// TIA Portal V16 export
// export: Created 2022-02-11T14:39:19.0580215Z, ExportSetting WithDefaults, DisplayName Totally Integrated Automation Portal, DisplayVersion V16 Update 1, DisplayName TIA Portal Version Control Interface, DisplayVersion V16, DisplayName TIA Portal Openness, DisplayVersion V16, DisplayName SINAMICS Startdrive Advanced, DisplayVersion V16 Update 5, DisplayName SINAMICS Startdrive G130, G150, S120, S150, SINAMICS MV, S210, DisplayVersion V16 Update 5, DisplayName SINAMICS Startdrive G110M, G120, G120C, G120D, G120P, G115D, DisplayVersion V16 Update 5, DisplayName STEP 7 Professional, DisplayVersion V16, DisplayName STEP 7 Safety, DisplayVersion V16, DisplayName WinCC Advanced, DisplayVersion V16, DisplayName SIMATIC Visualization Architect, DisplayVersion V16
ORGANIZATION_BLOCK "Main"   // OB1, LAD, ProgramCycle
TITLE = "Main Program Sweep (Cycle)"
VERSION : 0.1
// stored: IsIECCheckEnabled false
   VAR_TEMP
      OB1_EV_CLASS : Byte;   // Bits 0-3 = 1 (Coming event), Bits 4-7 = 1 (Event class 1)
      OB1_SCAN_1 : Byte;   // 1 (Cold restart scan 1 of OB 1), 3 (Scan 2-n of OB 1)
      OB1_PRIORITY : Byte;   // Priority of OB Execution
      OB1_OB_NUMBR : Byte;   // 1 (Organization block 1, OB1)
      OB1_RESERVED_1 : Byte;   // Reserved for system
      OB1_RESERVED_2 : Byte;   // Reserved for system
      BoardPosition : Int;   // Позиция подвижного борта
      OB1_PREV_CYCLE : Int;   // Cycle time of previous OB1 scan (milliseconds)
      OB1_MIN_CYCLE : Int;   // Minimum cycle time of OB1 (milliseconds)
      OB1_MAX_CYCLE : Int;   // Maximum cycle time of OB1 (milliseconds)
      OB1_DATE_TIME : Date_And_Time;   // Date and time OB1 started
   END_VAR
   VAR_TEMP   // added for the SCL form of the ladder/FBD networks
      _w1 : Bool;
      _w2 : Bool;
      _w3 : Bool;
      _s5time1 : S5Time;
   END_VAR
BEGIN

REGION Network 1: ProcessInput
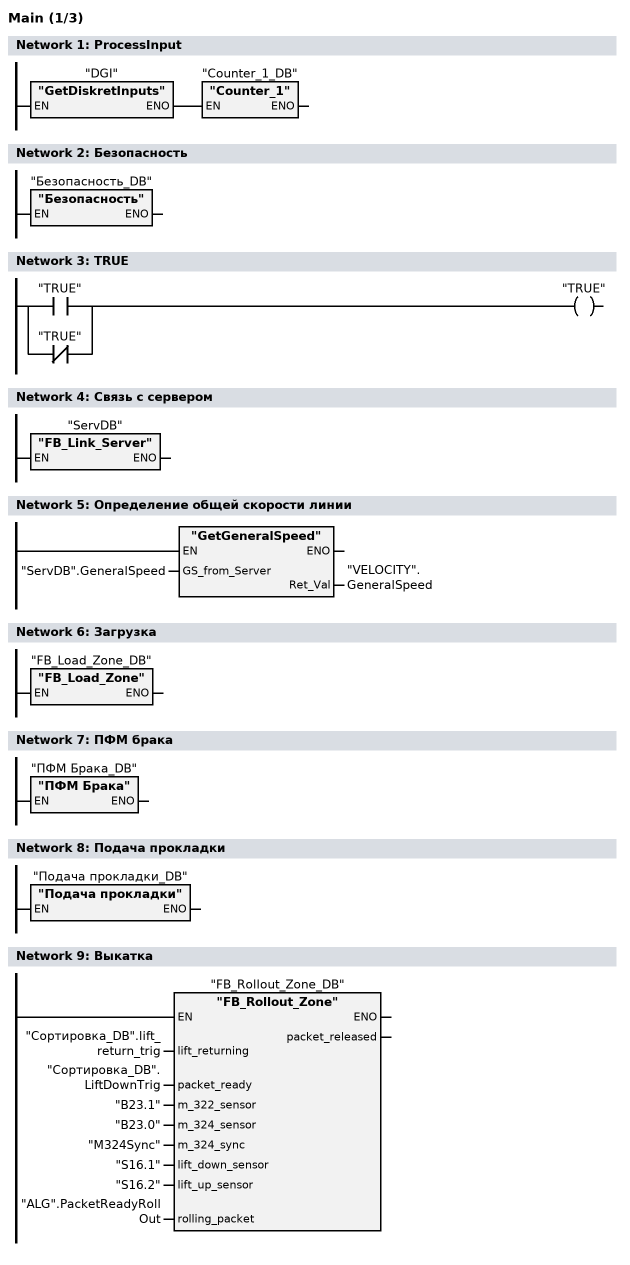
   RUNG wire#powerrail
      "DGI"()
      "Counter_1_DB"()
   END_RUNG
   // the same network as SCL:
   "DGI"(ENO => #_w1);   // "GetDiskretInputs"
   IF #_w1 THEN
       "Counter_1_DB"();   // "Counter_1"
   END_IF;
END_REGION

REGION Network 2: Безопасность
   RUNG wire#powerrail
      "Безопасность_DB"()
   END_RUNG
   // the same network as SCL:
   "Безопасность_DB"();   // "Безопасность"
END_REGION

REGION Network 3: TRUE
   RUNG wire#powerrail
      Contact( "TRUE" )
      wire#w1
      Coil( "TRUE" )
   END_RUNG
   RUNG wire#powerrail
      I_Contact( "TRUE" )
   END_RUNG wire#w1
   // the same network as SCL:
   "TRUE" := "TRUE" OR NOT "TRUE";
END_REGION

REGION Network 4: Связь с сервером
   RUNG wire#powerrail
      "ServDB"()
   END_RUNG
   // the same network as SCL:
   "ServDB"();   // "FB_Link_Server"
END_REGION

REGION Network 5: Определение общей скорости линии
   RUNG wire#powerrail
      "GetGeneralSpeed"(GS_from_Server := "ServDB".GeneralSpeed, Ret_Val => "VELOCITY".GeneralSpeed)
   END_RUNG
   // the same network as SCL:
   "VELOCITY".GeneralSpeed := "GetGeneralSpeed"(GS_from_Server := "ServDB".GeneralSpeed);
END_REGION

REGION Network 6: Загрузка
   RUNG wire#powerrail
      "FB_Load_Zone_DB"()
   END_RUNG
   // the same network as SCL:
   "FB_Load_Zone_DB"();   // "FB_Load_Zone"
END_REGION

REGION Network 7: ПФМ брака
   RUNG wire#powerrail
      "ПФМ Брака_DB"()
   END_RUNG
   // the same network as SCL:
   "ПФМ Брака_DB"();   // "ПФМ Брака"
END_REGION

REGION Network 8: Подача прокладки
   RUNG wire#powerrail
      "Подача прокладки_DB"()
   END_RUNG
   // the same network as SCL:
   "Подача прокладки_DB"();   // "Подача прокладки"
END_REGION

REGION Network 9: Выкатка
   RUNG wire#powerrail
      "FB_Rollout_Zone_DB"(lift_returning := "Сортировка_DB".lift_return_trig, packet_ready := "Сортировка_DB".LiftDownTrig, m_322_sensor := "B23.1", m_324_sensor := "B23.0", m_324_sync := "M324Sync", lift_down_sensor := "S16.1", lift_up_sensor := "S16.2", rolling_packet := "ALG".PacketReadyRollOut, packet_released =>)
   END_RUNG
   // the same network as SCL:
   "FB_Rollout_Zone_DB"(lift_returning := "Сортировка_DB".lift_return_trig,   // "FB_Rollout_Zone"
                        packet_ready := "Сортировка_DB".LiftDownTrig,
                        m_322_sensor := "B23.1",
                        m_324_sensor := "B23.0",
                        m_324_sync := "M324Sync",
                        lift_down_sensor := "S16.1",
                        lift_up_sensor := "S16.2",
                        rolling_packet := "ALG".PacketReadyRollOut);
END_REGION

REGION Network 10: Карусель прокладок
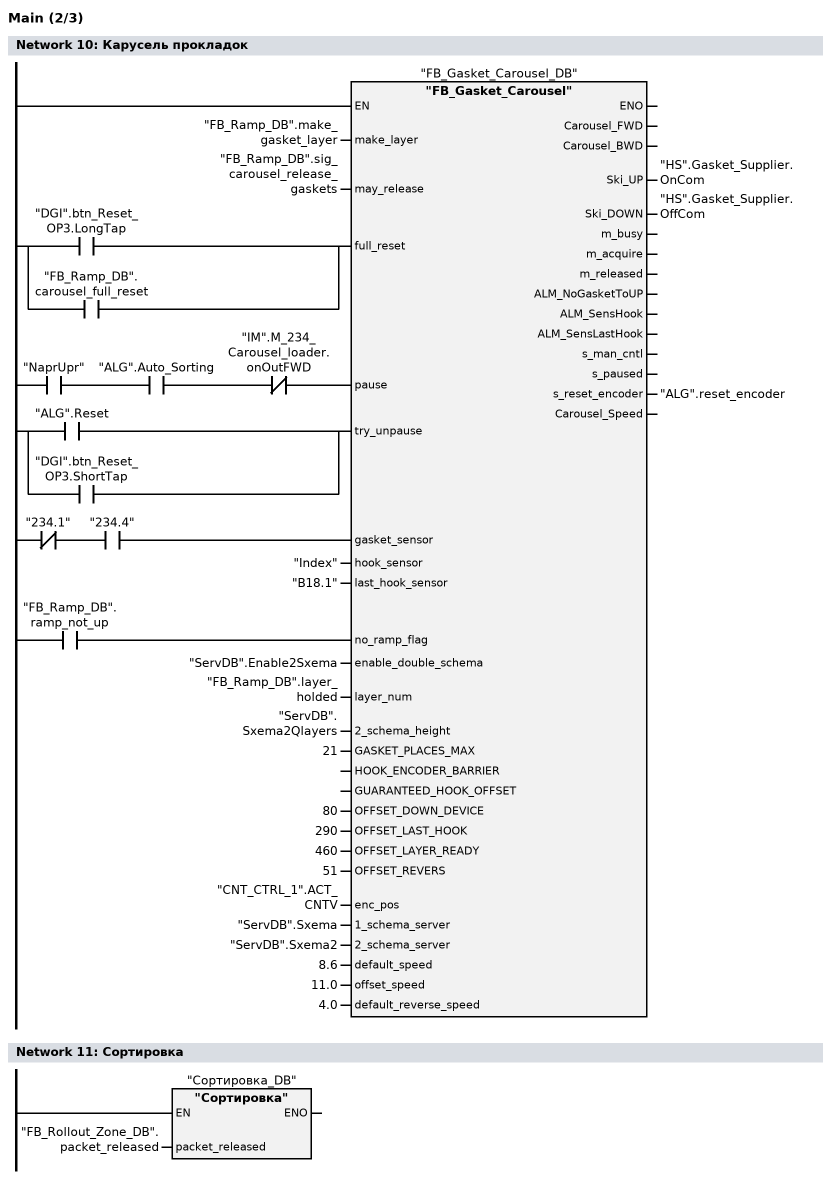
   RUNG wire#powerrail
      "FB_Gasket_Carousel_DB"(full_reset := wire#w1, pause := wire#w2, try_unpause := wire#w3, gasket_sensor := wire#w4, no_ramp_flag := wire#w5, make_layer := "FB_Ramp_DB".make_gasket_layer, may_release := "FB_Ramp_DB".sig_carousel_release_gaskets, hook_sensor := "Index", last_hook_sensor := "B18.1", enable_double_schema := "ServDB".Enable2Sxema, layer_num := "FB_Ramp_DB".layer_holded, "2_schema_height" := "ServDB".Sxema2Qlayers, GASKET_PLACES_MAX := 21, HOOK_ENCODER_BARRIER :=, GUARANTEED_HOOK_OFFSET :=, OFFSET_DOWN_DEVICE := 80, OFFSET_LAST_HOOK := 290, OFFSET_LAYER_READY := 460, OFFSET_REVERS := 51, enc_pos := "CNT_CTRL_1".ACT_CNTV, "1_schema_server" := "ServDB".Sxema, "2_schema_server" := "ServDB".Sxema2, default_speed := 8.6, offset_speed := 11.0, default_reverse_speed := 4.0, Carousel_FWD =>, Carousel_BWD =>, Ski_UP => "HS".Gasket_Supplier.OnCom, Ski_DOWN => "HS".Gasket_Supplier.OffCom, m_busy =>, m_acquire =>, m_released =>, ALM_NoGasketToUP =>, ALM_SensHook =>, ALM_SensLastHook =>, s_man_cntl =>, s_paused =>, s_reset_encoder => "ALG".reset_encoder, Carousel_Speed =>)
   END_RUNG
   RUNG wire#powerrail
      Contact( "DGI".btn_Reset_OP3.LongTap )
   END_RUNG wire#w1
   RUNG wire#powerrail
      Contact( "FB_Ramp_DB".carousel_full_reset )
   END_RUNG wire#w1
   RUNG wire#powerrail
      Contact( "NaprUpr" )
      Contact( "ALG".Auto_Sorting )
      I_Contact( "IM".M_234_Carousel_loader.onOutFWD )
   END_RUNG wire#w2
   RUNG wire#powerrail
      Contact( "ALG".Reset )
   END_RUNG wire#w3
   RUNG wire#powerrail
      Contact( "DGI".btn_Reset_OP3.ShortTap )
   END_RUNG wire#w3
   RUNG wire#powerrail
      I_Contact( "234.1" )
      Contact( "234.4" )
   END_RUNG wire#w4
   RUNG wire#powerrail
      Contact( "FB_Ramp_DB".ramp_not_up )
   END_RUNG wire#w5
   // the same network as SCL:
   "FB_Gasket_Carousel_DB"(make_layer := "FB_Ramp_DB".make_gasket_layer,   // "FB_Gasket_Carousel"
                           may_release := "FB_Ramp_DB".sig_carousel_release_gaskets,
                           full_reset := "DGI".btn_Reset_OP3.LongTap OR "FB_Ramp_DB".carousel_full_reset,
                           pause := "NaprUpr" AND "ALG".Auto_Sorting AND NOT "IM".M_234_Carousel_loader.onOutFWD,
                           try_unpause := "ALG".Reset OR "DGI".btn_Reset_OP3.ShortTap,
                           gasket_sensor := NOT "234.1" AND "234.4",
                           hook_sensor := "Index",
                           last_hook_sensor := "B18.1",
                           no_ramp_flag := "FB_Ramp_DB".ramp_not_up,
                           enable_double_schema := "ServDB".Enable2Sxema,
                           layer_num := "FB_Ramp_DB".layer_holded,
                           "2_schema_height" := "ServDB".Sxema2Qlayers,
                           GASKET_PLACES_MAX := 21,
                           OFFSET_DOWN_DEVICE := 80,
                           OFFSET_LAST_HOOK := 290,
                           OFFSET_LAYER_READY := 460,
                           OFFSET_REVERS := 51,
                           enc_pos := "CNT_CTRL_1".ACT_CNTV,
                           "1_schema_server" := "ServDB".Sxema,
                           "2_schema_server" := "ServDB".Sxema2,
                           default_speed := 8.6,
                           offset_speed := 11.0,
                           default_reverse_speed := 4.0,
                           Ski_UP => "HS".Gasket_Supplier.OnCom,
                           Ski_DOWN => "HS".Gasket_Supplier.OffCom,
                           s_reset_encoder => "ALG".reset_encoder);
END_REGION

REGION Network 11: Сортировка
   RUNG wire#powerrail
      "Сортировка_DB"(packet_released := "FB_Rollout_Zone_DB".packet_released)
   END_RUNG
   // the same network as SCL:
   "Сортировка_DB"(packet_released := "FB_Rollout_Zone_DB".packet_released);   // "Сортировка"
END_REGION

REGION Network 12: Авто режим подвижного борта
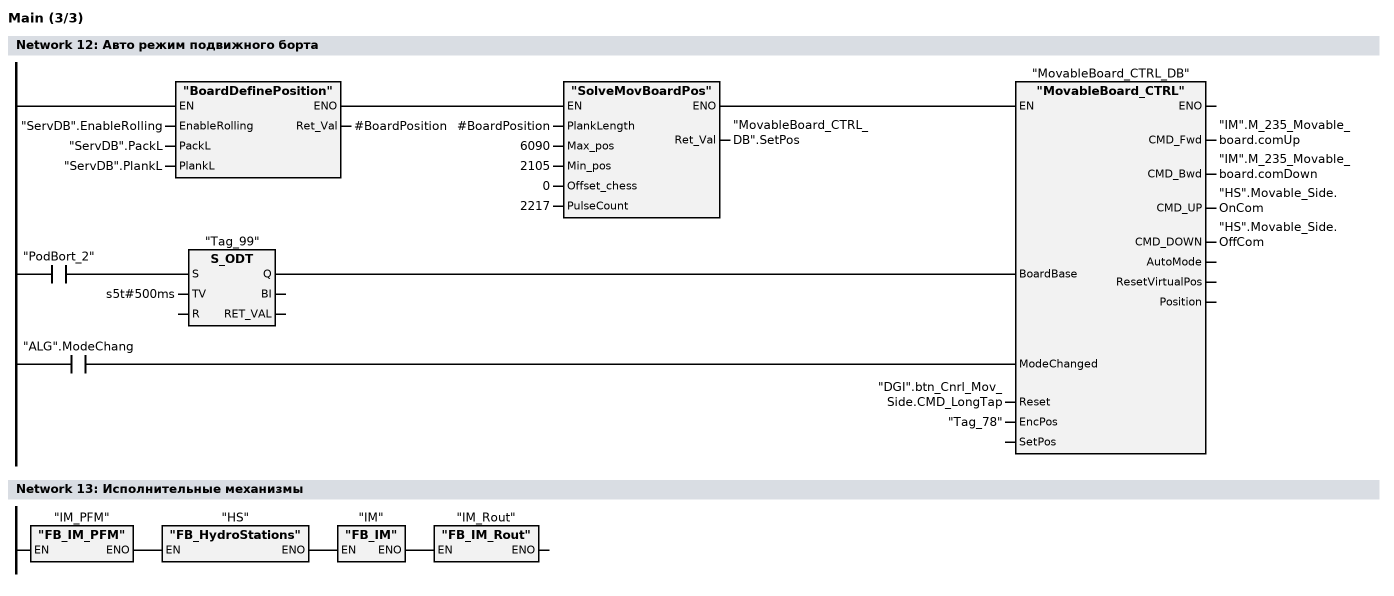
   RUNG wire#powerrail
      "BoardDefinePosition"(EnableRolling := "ServDB".EnableRolling, PackL := "ServDB".PackL, PlankL := "ServDB".PlankL, Ret_Val => #BoardPosition)
      "SolveMovBoardPos"(PlankLength := #BoardPosition, Max_pos := 6090, Min_pos := 2105, Offset_chess := 0, PulseCount := 2217, Ret_Val => "MovableBoard_CTRL_DB".SetPos)
      "MovableBoard_CTRL_DB"(BoardBase := wire#w1, ModeChanged := wire#w2, Reset := "DGI".btn_Cnrl_Mov_Side.CMD_LongTap, EncPos := "Tag_78", SetPos :=, CMD_Fwd => "IM".M_235_Movable_board.comUp, CMD_Bwd => "IM".M_235_Movable_board.comDown, CMD_UP => "HS".Movable_Side.OnCom, CMD_DOWN => "HS".Movable_Side.OffCom, AutoMode =>, ResetVirtualPos =>, Position =>)
   END_RUNG
   RUNG wire#powerrail
      Contact( "PodBort_2" )
      S_ODT(T_NO := "Tag_99", TV := s5t#500ms, R :=, BI =>, RET_VAL =>)
   END_RUNG wire#w1
   RUNG wire#powerrail
      Contact( "ALG".ModeChang )
   END_RUNG wire#w2
   // the same network as SCL:
   #BoardPosition := "BoardDefinePosition"(EnableRolling := "ServDB".EnableRolling,
                           PackL := "ServDB".PackL,
                           PlankL := "ServDB".PlankL,
                           ENO => #_w1);
   "MovableBoard_CTRL_DB".SetPos := "SolveMovBoardPos"(EN := #_w1,
                           PlankLength := #BoardPosition,
                           Max_pos := 6090,
                           Min_pos := 2105,
                           Offset_chess := 0,
                           PulseCount := 2217,
                           ENO => #_w2);
   #_s5time1 := S_ODT(T_NO := "Tag_99", S := "PodBort_2", TV := s5t#500ms, Q => #_w3);
   IF #_w2 THEN
       "MovableBoard_CTRL_DB"(BoardBase := #_w3,   // "MovableBoard_CTRL"
                              ModeChanged := "ALG".ModeChang,
                              Reset := "DGI".btn_Cnrl_Mov_Side.CMD_LongTap,
                              EncPos := "Tag_78",
                              CMD_Fwd => "IM".M_235_Movable_board.comUp,
                              CMD_Bwd => "IM".M_235_Movable_board.comDown,
                              CMD_UP => "HS".Movable_Side.OnCom,
                              CMD_DOWN => "HS".Movable_Side.OffCom);
   END_IF;
END_REGION

REGION Network 13: Исполнительные механизмы
   RUNG wire#powerrail
      "IM_PFM"()
      "HS"()
      "IM"()
      "IM_Rout"()
   END_RUNG
   // the same network as SCL:
   "IM_PFM"(ENO => #_w1);   // "FB_IM_PFM"
   "HS"(EN := #_w1, ENO => #_w2);   // "FB_HydroStations"
   "IM"(EN := #_w2, ENO => #_w3);   // "FB_IM"
   IF #_w3 THEN
       "IM_Rout"();   // "FB_IM_Rout"
   END_IF;
END_REGION
END_ORGANIZATION_BLOCK
